PROGRAM POU
VAR
END_VAR

END_PROGRAM

(* stored: Version 1.1.0.1, ProductVersion 3.1.4024.12
   POU POU: Id {1a555e11-0331-42ea-99a9-05abce928c6a}, SpecialFunc None *)
